FUNCTION checkDistance : BOOL
VAR_INPUT
    distance_in_function : REAL;  // Distance from the mirror
END_VAR

// If the distance is less than or equal to 1 meter, return TRUE, else return FALSE
IF distance_in_function<= 1.0 THEN
    checkDistance := TRUE;
ELSE
    checkDistance := FALSE;
END_IF

END_FUNCTION

(* stored: Version 1.1.0.1, ProductVersion 3.1.4024.12
   POU checkDistance: Id {454bb1e2-994d-4bd1-9b0d-e3aea2c31f5b}, SpecialFunc None *)
